FUNCTION_BLOCK SS5a_ps_Raiser_n_Flipper (* Composite FB wrapping other FBs *)
  (* Standard: 61499-2 *)
  (* Version 1.0, 2025-08-26, PS_Transformer_for_Unknown *)
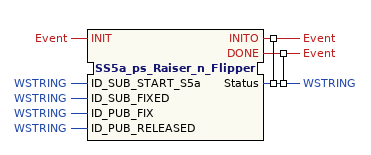
  EVENT_INPUT
    INIT; (* Initialization Request *)
  END_EVENT
  EVENT_OUTPUT
    INITO WITH Status; (* Initialization Confirm *)
    DONE WITH Status; (* Execution Confirmation *)
  END_EVENT
  VAR_INPUT
    ID_SUB_START_S5a : WSTRING;
    ID_SUB_FIXED : WSTRING;
    ID_PUB_FIX : WSTRING;
    ID_PUB_RELEASED : WSTRING;
  END_VAR
  VAR_OUTPUT
    Status : WSTRING; (* Output event qualifier *)
  END_VAR
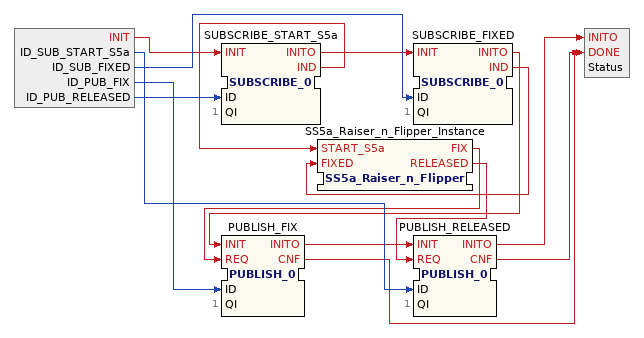
  FBS
    SS5a_Raiser_n_Flipper_Instance : SS5a_Raiser_n_Flipper;
    SUBSCRIBE_START_S5a : SUBSCRIBE_0(QI := 1);
    SUBSCRIBE_FIXED : SUBSCRIBE_0(QI := 1);
    PUBLISH_FIX : PUBLISH_0(QI := 1);
    PUBLISH_RELEASED : PUBLISH_0(QI := 1);
  END_FBS
  EVENT_CONNECTIONS
    INIT TO SUBSCRIBE_START_S5a.INIT;
    SUBSCRIBE_START_S5a.INITO TO SUBSCRIBE_FIXED.INIT;
    SUBSCRIBE_FIXED.INITO TO PUBLISH_FIX.INIT;
    PUBLISH_FIX.INITO TO PUBLISH_RELEASED.INIT;
    PUBLISH_RELEASED.INITO TO INITO;
    SUBSCRIBE_START_S5a.IND TO SS5a_Raiser_n_Flipper_Instance.START_S5a;
    SUBSCRIBE_FIXED.IND TO SS5a_Raiser_n_Flipper_Instance.FIXED;
    SS5a_Raiser_n_Flipper_Instance.FIX TO PUBLISH_FIX.REQ;
    SS5a_Raiser_n_Flipper_Instance.RELEASED TO PUBLISH_RELEASED.REQ;
    PUBLISH_FIX.CNF TO DONE;
    PUBLISH_RELEASED.CNF TO DONE;
  END_CONNECTIONS
  DATA_CONNECTIONS
    ID_SUB_START_S5a TO SUBSCRIBE_START_S5a.ID;
    ID_SUB_FIXED TO SUBSCRIBE_FIXED.ID;
    ID_PUB_FIX TO PUBLISH_FIX.ID;
    ID_PUB_RELEASED TO PUBLISH_RELEASED.ID;
  END_CONNECTIONS
END_FUNCTION_BLOCK
